(* IEC 61131-3 sources: GASR-FBE/bin/fad2/AppSemaforo, 10 files *)

(* ---- CAR_SEMAPHORE.st ---- *)
(* Generated by xml2st *)
FUNCTION_BLOCK CAR_SEMAPHORE
  EVENT_INPUT
    INIT;
    SET;
  END_EVENT
  EVENT_OUTPUT
    INIT0;
    OUT_RED;
    OUT_YELLOW;
    OUT_GREEN;
  END_EVENT

  EC_STATES
    RUN: ALG_RUN ->, -> OUT_RED, -> OUT_YELLOW, -> OUT_GREEN;
    START;
    INIT: ALG_INIT -> INIT0, -> OUT_RED, -> OUT_YELLOW, -> OUT_GREEN;
  END_STATES

  EC_TRANSITIONS
    START TO INIT := INIT;
    INIT TO START := 1;
    START TO RUN := SET;
    RUN TO START := 1;
  END_TRANSITIONS

  VAR_INPUT
    CYCLE: BYTE;
  END_VAR

  VAR_OUTPUT
    RED: BOOL;
    YELLOW: BOOL;
    GREEN: BOOL;
  END_VAR

  ALGORITHM ALG_RUN IN ST:
RED := 0; YELLOW := 0; GREEN := 0;     IF(CYCLE = 0) THEN    RED:=1; END_IF;    IF(CYCLE=1)THEN GREEN:=1; END_IF;   IF(CYCLE=2)THEN YELLOW:=1; END_IF;
  END_ALGORITHM

  ALGORITHM ALG_INIT IN ST:
 RED := 1; GREEN := 0; YELLOW := 0;
  END_ALGORITHM

END_FUNCTION_BLOCK

(* ---- E_SPLIT.st ---- *)
(* Generated by xml2st *)
FUNCTION_BLOCK E_SPLIT
  EVENT_INPUT
    EI1;
  END_EVENT
  EVENT_OUTPUT
    EO1;
    EO2;
  END_EVENT

  EC_STATES
    RUN: -> EO1, -> EO2;
    START;
  END_STATES

  EC_TRANSITIONS
    START TO RUN := EI1;
    RUN TO START := 1;
  END_TRANSITIONS

  VAR_INPUT
  END_VAR

  VAR_OUTPUT
  END_VAR

END_FUNCTION_BLOCK

(* ---- IO_READER.st ---- *)
(* Generated by xml2st *)
FUNCTION_BLOCK IO_READER
  EVENT_INPUT
    INIT;
    RSP;
  END_EVENT
  EVENT_OUTPUT
    INIT0;
    IND;
  END_EVENT

  EC_STATES
    START;
    READ: ALG_READ -> IND;
    INIT: ALG_INIT -> INIT0;
  END_STATES

  EC_TRANSITIONS
    START TO INIT := INIT;
    INIT TO START := 1;
    START TO READ := RSP;
    READ TO START := 1;
  END_TRANSITIONS

  VAR_INPUT
    QI: BOOL;
    PARAMS: BYTE;
    SD_1: BYTE;
  END_VAR

  VAR_OUTPUT
    QO: BOOL;
    STATUS: BOOL;
    RD_1: BYTE;
  END_VAR

  ALGORITHM ALG_INIT IN ST:

  END_ALGORITHM

  ALGORITHM ALG_READ IN ST:
RD_1 := GET_REG(SD_1);
  END_ALGORITHM

END_FUNCTION_BLOCK

(* ---- IO_WRITER.st ---- *)
(* Generated by xml2st *)
FUNCTION_BLOCK IO_WRITER
  EVENT_INPUT
    INIT;
    REQ;
  END_EVENT
  EVENT_OUTPUT
    INIT0;
    CNF;
  END_EVENT

  EC_STATES
    WRITE: ALG_WRITE -> CNF;
    START;
    INIT: ALG_INIT -> INIT0;
  END_STATES

  EC_TRANSITIONS
    START TO INIT := INIT;
    INIT TO START := 1;
    START TO WRITE := REQ;
    WRITE TO START := 1;
  END_TRANSITIONS

  VAR_INPUT
    QI: BOOL;
    PARAMS: BYTE;
    SD_1: BYTE;
    SD_2: BYTE;
  END_VAR

  VAR_OUTPUT
    QO: BOOL;
    STATUS: BYTE;
    RD_1: BYTE;
  END_VAR

  ALGORITHM ALG_WRITE IN ST:
SET_REG(SD_1, SD_2);
  END_ALGORITHM

  ALGORITHM ALG_INIT IN ST:

  END_ALGORITHM

END_FUNCTION_BLOCK

(* ---- PUB_2.st ---- *)
(* Generated by xml2st *)
FUNCTION_BLOCK PUB_2
  EVENT_INPUT
    INIT;
    REQ;
  END_EVENT
  EVENT_OUTPUT
    INIT0;
  END_EVENT

  EC_STATES
    START;
    SEND: ALG_SND ->;
    INIT: ALG_INIT -> INIT0;
  END_STATES

  EC_TRANSITIONS
    START TO INIT := INIT;
    START TO SEND := REQ;
    SEND TO START := 1;
    INIT TO START := 1;
  END_TRANSITIONS

  VAR_INPUT
    ID: BYTE;
    RD_1: BYTE;
    RD_2: BOOL;
  END_VAR

  VAR_OUTPUT
  END_VAR

  VAR
    RD_1_: BYTE;
    RD_2_: BOOL;
  END_VAR

  ALGORITHM ALG_SND IN ST:
    IF (NOT(RD_1_ = RD_1)) OR (NOT(RD_2_ = RD_2)) THEN
      ASM
	    LOAD RD_1
	    LOAD RD_2
	    CONST 2
	    LOAD ID
	    NISND
	  END_ASM
	  RD_1_ := RD_1;
	  RD_2_ := RD_2;
	END_IF;
  END_ALGORITHM

  ALGORITHM ALG_INIT IN ST:

  END_ALGORITHM

END_FUNCTION_BLOCK

(* ---- SEM_CONTROL.st ---- *)
(* Generated by xml2st *)
FUNCTION_BLOCK SEM_CONTROL
  EVENT_INPUT
    INIT;
    ETIME;
    BTWALKER;
  END_EVENT
  EVENT_OUTPUT
    INIT0;
    SET_SEMAPHORE;
  END_EVENT

  EC_STATES
    START;
    RUN: ALG_RUN -> SET_SEMAPHORE;
    ST_WALKER: ALG_WALKER ->;
    INIT: ALG_INIT -> INIT0;
  END_STATES

  EC_TRANSITIONS
    START TO INIT := INIT;
    START TO RUN := ETIME;
    INIT TO START := 1;
    RUN TO START := 1;
    START TO ST_WALKER := BTWALKER;
    ST_WALKER TO START := 1;
  END_TRANSITIONS

  VAR_INPUT
    lbtwalker: BOOL;
    btwalker: BOOL;
  END_VAR

  VAR_OUTPUT
    SEMAPHORE_1: BYTE;
    SEMAPHORE_2: BYTE;
    SEMAPHORE_3: BYTE;
    SEMAPHORE_4: BYTE;
    WALKER: BOOL;
  END_VAR

  ALGORITHM ALG_INIT IN ST:
SEMAPHORE_1 := 0; SEMAPHORE_2 := 0; SEMAPHORE_3 := 0; SEMAPHORE_4 := 0; WALKER :=0;
  END_ALGORITHM

  ALGORITHM ALG_WALKER IN ST:
IF(btwalker) THEN lbtwalker:=1; END_IF;
  END_ALGORITHM

  ALGORITHM ALG_RUN IN ST:
IF(WALKER) THEN  WALKER := 0;  SEMAPHORE_1 := 1;     SEMAPHORE_2 := 0;   lbtwalker := 0; ELSE  IF(SEMAPHORE_2 = 0) THEN     SEMAPHORE_1 := SEMAPHORE_1 + 1;     IF(SEMAPHORE_1 >= 3) THEN       SEMAPHORE_1 := 0;       SEMAPHORE_2 := 1;     END_IF;   ELSE     SEMAPHORE_2 := SEMAPHORE_2 + 1;     IF(SEMAPHORE_2 >= 3) THEN      IF(lbtwalker) THEN         WALKER := 1;     SEMAPHORE_1 := 0;        SEMAPHORE_2 := 0;     ELSE     SEMAPHORE_1 := 1;        SEMAPHORE_2 := 0;     END_IF;   END_IF;    END_IF;  END_IF;
  END_ALGORITHM

END_FUNCTION_BLOCK

(* ---- SUB_2.st ---- *)
(* Generated by xml2st *)
FUNCTION_BLOCK SUB_2
  EVENT_INPUT
    INIT;
  END_EVENT
  EVENT_OUTPUT
    INIT0;
    RSP;
  END_EVENT

  EC_STATES
    START;
    RCV: ALG_RCV -> RSP;
    INIT: ALG_INIT -> INIT0;
  END_STATES

  EC_TRANSITIONS
    START TO INIT := INIT;
    INIT TO START := 1;
    START TO RCV := 1;
    RCV TO START := 1;
  END_TRANSITIONS

  VAR_INPUT
    ID: BYTE;
  END_VAR

  VAR_OUTPUT
    SD_1: BYTE;
    SD_2: BOOL;
  END_VAR

  ALGORITHM ALG_RCV IN ST:
	ASM
		CONST 2
		LOAD ID
		NIRCV
		IF GOTO process
		GOTO out
	process:
		STORE SD_1
		STORE SD_2
	out:
	END_ASM
  END_ALGORITHM

  ALGORITHM ALG_INIT IN ST:

  END_ALGORITHM

END_FUNCTION_BLOCK

(* ---- E_CYCLE.st ---- *)
CUSTOM FUNCTION_BLOCK E_CYCLE
	EVENT_INPUT
		START;
		STOP;
	END_EVENT

	EVENT_OUTPUT
		EO;
	END_EVENT

	VAR_INPUT
		DT:BYTE;
	END_VAR

	VAR
		oldt: BYTE;
		count:BYTE;
		state: BYTE;
	END_VAR

	ALGORITHM ALG_INIT:
		oldt := GET_REG(100);
		count := 0;
		state := 0;
		EO:=0;
	END_ALGORITHM
	ALGORITHM ALG_RUN:
		IF(START) THEN
			state :=1;
			START := 0;
			count := 0;
			oldt := GET_REG(100);
		END_IF;
		IF(STOP)THEN
			state := 0;
			EO := 0;
		END_IF;
		(*
		IF(EO) THEN
			EO := 0;
		END_IF;
		*)
		IF(state = 1) THEN
			IF(NOT (oldt = GET_REG(100))) THEN
				count := count + 1;
				IF(count = DT) THEN
					EO := 1;
					count := 0;
				END_IF;
				oldt := GET_REG(100);
			END_IF;
		END_IF;
	END_ALGORITHM

END_FUNCTION_BLOCK

(* ---- SEM_CONTROL-ALG_RUN.st ---- *)
IF(WALKER) THEN
	WALKER := 0;
	SEMAPHORE_1 := 1;
	SEMAPHORE_2 := 0;
	lbtwalker := 0;
ELSE
	IF(SEMAPHORE_2 = 0) THEN
		SEMAPHORE_1 := SEMAPHORE_1 + 1;
		IF(SEMAPHORE_1 >= 3) THEN
			SEMAPHORE_1 := 0;
			SEMAPHORE_2 := 1;
		END_IF;
	ELSE
		SEMAPHORE_2 := SEMAPHORE_2 + 1;
		IF(SEMAPHORE_2 >= 3) THEN
			IF(lbtwalker) THEN
				WALKER := 1;
				SEMAPHORE_1 := 0;
				SEMAPHORE_2 := 0;
			ELSE
				SEMAPHORE_1 := 1;
				SEMAPHORE_2 := 0;
			END_IF;
		END_IF;
	END_IF;
END_IF;

(*
IF(SEMAPHORE_2 = 0) THEN  SEMAPHORE_1 := SEMAPHORE_1 + 1;  IF(SEMAPHORE_1 >= 3) THEN   SEMAPHORE_1 := 0;   SEMAPHORE_2 := 1;  END_IF; ELSE  SEMAPHORE_2 := SEMAPHORE_2 + 1;  IF(SEMAPHORE_2 >= 3) THEN   SEMAPHORE_1 := 1;   SEMAPHORE_2 := 0;  END_IF;  END_IF; R:=2.3 + 4.5; R:=(R+1.2)*3.0; R := R/2.0;
*)

(* ---- START.st ---- *)
CUSTOM FUNCTION_BLOCK START

	EVENT_OUTPUT
		COLD;
		STOP;
	END_EVENT

	ALGORITHM ALG_INIT:
		COLD:=1;
	END_ALGORITHM
	ALGORITHM ALG_RUN:

	END_ALGORITHM

END_FUNCTION_BLOCK
